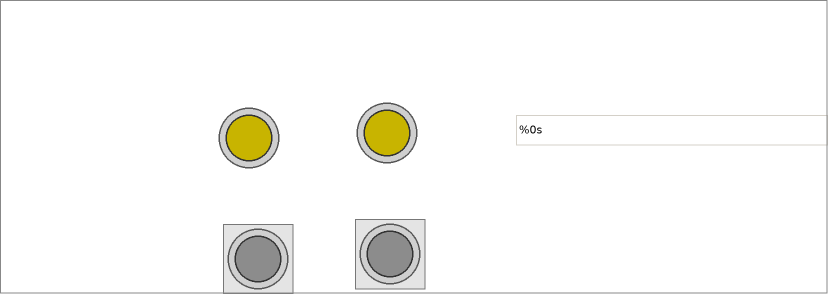
VISUALIZATION Visualization  // 828x294
    Lamp1 (214,103 70x70), variable: MAIN.test_output[0], style: Lamp-Lamp1-Yellow
    PushSwitch (223,224 70x70), variable: MAIN.test_input[0], behaviour: TAP, style: Switch-PushSwitch-Gray
    Lamp1 (352,98 70x70), variable: MAIN.test_output[1], style: Lamp-Lamp1-Yellow
    PushSwitch (355,219 70x70), variable: MAIN.test_input[1], behaviour: TOGGLE, style: Switch-PushSwitch-Gray
    Textfield (516,115 312x30), "%0s", text variable: MAIN.test_string
        OnMouseClick: write the text variable via Edit
END_VISUALIZATION

(* stored: Version 1.1.0.1, ProductVersion 3.1.4024.12
   Visu Visualization: Id {70d9ba4e-a4bc-4a02-8550-556a38b71399} *)
